FUNCTION_BLOCK TwoCylDiscr
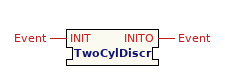
  EVENT_INPUT
    INIT;
  END_EVENT
  EVENT_OUTPUT
    INITO;
  END_EVENT
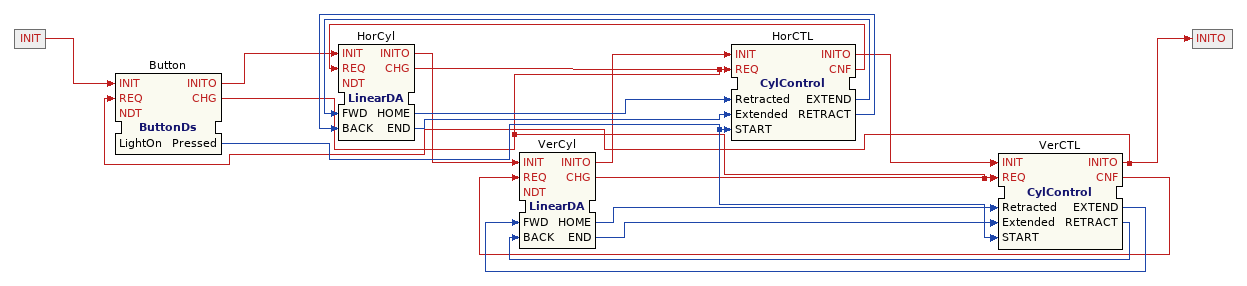
  FBS
    HorCTL : CylControl;
    VerCTL : CylControl;
    Button : ButtonDs;
    HorCyl : LinearDA;
    VerCyl : LinearDA;
  END_FBS
  EVENT_CONNECTIONS
    Button.INITO TO HorCyl.INIT;
    HorCyl.INITO TO VerCyl.INIT;
    VerCyl.INITO TO HorCTL.INIT;
    HorCTL.CNF TO HorCyl.REQ;
    HorCyl.CHG TO HorCTL.REQ;
    VerCyl.CHG TO VerCTL.REQ;
    HorCTL.INITO TO VerCTL.INIT;
    VerCTL.CNF TO VerCyl.REQ;
    Button.CHG TO VerCTL.REQ;
    INIT TO Button.INIT;
    VerCTL.INITO TO INITO;
    Button.CHG TO HorCTL.REQ;
    VerCTL.INITO TO Button.REQ;
  END_CONNECTIONS
  DATA_CONNECTIONS
    HorCyl.HOME TO HorCTL.Retracted;
    HorCyl.END TO HorCTL.Extended;
    Button.Pressed TO HorCTL.START;
    HorCTL.EXTEND TO HorCyl.FWD;
    HorCTL.RETRACT TO HorCyl.BACK;
    VerCyl.HOME TO VerCTL.Retracted;
    VerCyl.END TO VerCTL.Extended;
    VerCTL.RETRACT TO VerCyl.BACK;
    VerCTL.EXTEND TO VerCyl.FWD;
    Button.Pressed TO VerCTL.START;
  END_CONNECTIONS
END_FUNCTION_BLOCK
